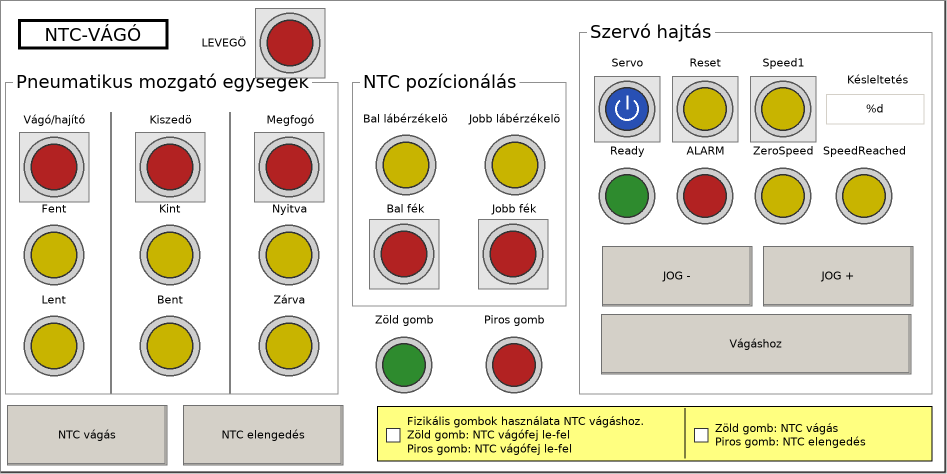
VISUALIZATION NTC_szerviz  // 947x474
    Rectangle (0,0 945x472)
    GroupBox (579,24 353x370), "Szervó hajtás"
        Lamp1 (15,139 66x66), variable: NTC.bReady, style: Lamp-Lamp1-Green
        Lamp1 (93,139 66x66), variable: NTC.bAlarm, style: Lamp-Lamp1-Red
        PowerSwitch (15,52 66x66), variable: NTC.bServoON, behaviour: TOGGLE, style: Switch-PowerSwitch-Blue
        PushSwitch (93,52 66x66), variable: NTC.bReset, behaviour: TOGGLE, style: Switch-PushSwitch-Yellow
        Lamp1 (171,139 66x66), variable: NTC.bZeroSpeed, style: Lamp-Lamp1-Yellow
        Label (170,112 69x30), "ZeroSpeed"
        Lamp1 (252,139 66x66), variable: NTC.bSpeedReached, style: Lamp-Lamp1-Yellow
        Label (239,112 93x30), "SpeedReached"
        PushSwitch (171,52 66x66), variable: NTC.bSpeed1, behaviour: TOGGLE, style: Switch-PushSwitch-Yellow
        Label (170,24 69x30), "Speed1"
        Button (184,222 150x60), "JOG +"
            tap NTC.bJogPlus
        Button (23,222 150x60), "JOG -"
            tap NTC.bJogMinus
        Textfield (247,70 98x30), "%d", text variable: NTC.iDelayFor
            OnMouseClick: write the text variable via VisuDialogs.Numpad, min -10000, max -1
        Label (264,41 69x30), "Késleltetés"
        Button (22,290 310x60), "Vágáshoz"
            OnMouseClick: execute { NTC.bVagashoz:=TRUE; }
        Label (14,24 69x30), "Servo"
        Label (92,24 69x30), "Reset"
        Label (14,112 69x30), "Ready"
        Label (92,112 69x30), "ALARM"
    GroupBox (5,74 333x320), "Pneumatikus mozgató egységek"
        PushSwitch (14,58 70x70), variable: NTCProcess.bVagoHajlito, behaviour: TOGGLE, style: Switch-PushSwitch-Red
        Label (15,31 69x30), "Vágó/hajító"
        Lamp1 (14,237 70x70), variable: NTCProcess.bVagoHajlitoLent, style: Lamp-Lamp1-Yellow
        Label (27,211 44x30), "Lent"
        Lamp1 (14,146 70x70), variable: NTCProcess.bVagoHajlitoFent, style: Lamp-Lamp1-Yellow
        Label (24,120 50x30), "Fent"
        Label (131,31 69x30), "Kiszedö"
        Lamp1 (130,237 70x70), variable: NTCProcess.bKiszedoBent, style: Lamp-Lamp1-Yellow
        Label (146,211 38x30), "Bent"
        Lamp1 (130,146 70x70), variable: NTCProcess.bKiszedoKint, style: Lamp-Lamp1-Yellow
        Label (147,120 36x30), "Kint"
        PushSwitch (130,58 70x70), variable: NTCProcess.bKiszedo, behaviour: TOGGLE, style: Switch-PushSwitch-Red
        PushSwitch (249,58 70x70), variable: NTCProcess.bMegfogo, behaviour: TOGGLE, style: Switch-PushSwitch-Red
        Lamp1 (249,237 70x70), variable: NTCProcess.bMegfogoZarva, style: Lamp-Lamp1-Yellow
        Label (265,211 39x30), "Zárva"
        Lamp1 (249,146 70x70), variable: NTCProcess.bMegfogoNyitva, style: Lamp-Lamp1-Yellow
        Label (261,120 47x30), "Nyitva"
        Label (251,31 69x30), "Megfogó"
        Line (106,319) (106,38)
        Line (225,319) (225,38)
    RoundedRectangle (18,19 150x30)
    Label (18,20 150x30), "NTC-VÁGÓ"
    Group (194,8 131x70)
        PushSwitch (61,0 70x70), variable: MAIN.bLevego, behaviour: TOGGLE, style: Switch-PushSwitch-Red
        Label (0,20 55x30), "LEVEGÖ"
    Button (7,405 160x60), "NTC vágás"
        OnMouseClick: execute { NTCProcess.s_InCommand:='VAGAS'; }
    Button (183,405 160x60), "NTC elengedés"
        OnMouseClick: execute { NTCProcess.s_InCommand:='NTC_ELENGED'; }
    Rectangle (377,406 555x55)
    Checkbox (692,413 227x44), "Zöld gomb: NTC vágás Piros gomb: NTC elengedés", variable: NTC.bVagasGombbal, input disabled if: NTC.bVagoFelLeGombbal AND FALSE
    GroupBox (352,74 214x232), "NTC pozícionálás"
        Label (19,125 69x20), "Bal fék"
        Lamp1 (19,56 70x70), variable: NTC.bNTCLaberzekeloBal, style: Lamp-Lamp1-Yellow
        Label (4,35 99x20), "Bal lábérzékelö"
        PushSwitch (126,145 70x70), variable: NTC.bNTCFekJobb, behaviour: TOGGLE, style: Switch-PushSwitch-Red
    PushSwitch (369,219 70x70), variable: NTC.bNTCFekBal, behaviour: TOGGLE, style: Switch-PushSwitch-Red
    Label (480,199 69x20), "Jobb fék"
    Lamp1 (480,130 70x70), variable: NTC.bNTCLaberzekeloJobb, style: Lamp-Lamp1-Yellow
    Label (465,109 99x20), "Jobb lábérzékelö"
    Lamp1 (371,332 66x66), variable: NTC.bZoldGomb, style: Lamp-Lamp1-Green
    Lamp1 (481,332 66x66), variable: NTC.bPirosGomb, style: Lamp-Lamp1-Red
    Label (480,310 69x20), "Piros gomb"
    Label (370,310 69x20), "Zöld gomb"
    Checkbox (384,413 297x44), "Fizikális gombok használata NTC vágáshoz. Zöld gomb: NTC vágófej le-fel Piros gomb: NTC vágófej le-fel", variable: NTC.bVagoFelLeGombbal, input disabled if: TRUE
    Line (685,458) (685,408)
END_VISUALIZATION

(* stored: Version 1.1.0.1, ProductVersion 3.1.4024.11
   Visu NTC_szerviz: Id {4411d55a-3928-4364-bbbf-5d98ed552431} *)
